Fanuc TP program (LS listing): _rs_s_retreat.ls

/PROG  _RS_S_RETREAT
/ATTR
OWNER		= MNEDITOR;
COMMENT		= "";
PROG_SIZE	= 309;
CREATE		= DATE 21-08-19  TIME 21:16:20;
MODIFIED	= DATE 21-08-19  TIME 21:16:20;
FILE_NAME	= _LS_S_RE;
VERSION		= 0;
LINE_COUNT	= 6;
MEMORY_SIZE	= 657;
PROTECT		= READ_WRITE;
TCD:  STACK_SIZE	= 0,
      TASK_PRIORITY	= 50,
      TIME_SLICE	= 0,
      BUSY_LAMP_OFF	= 0,
      ABORT_REQUEST	= 0,
      PAUSE_REQUEST	= 0;
DEFAULT_GROUP	= 1,*,*,*,*;
CONTROL_CODE	= 00000000 00000000;
/APPL
/APPL

AUTO_SINGULARITY_HEADER;
  ENABLE_SINGULARITY_AVOIDANCE   : TRUE;
/MN
   1:  OVERRIDE=R[1:Override Speed] ;
   2:  PR[11:SAND OFFSET]=LPOS    ;
   3:  R[66:S RS HOLDER]=PR[11,3:SAND OFFSET]    ;
   4:  R[66:S RS HOLDER]=R[66:S RS HOLDER]+R[14:RETREAT UP]    ;
   5:  PR[11,3:SAND OFFSET]=R[66:S RS HOLDER]    ;
   6:L PR[11:SAND OFFSET] 100mm/sec CNT100    ;
/POS
/END
